FUNCTION_BLOCK WOOD_COUNTER
  {SET_ATTRIBUTE(OpcUa, SERVICE)}
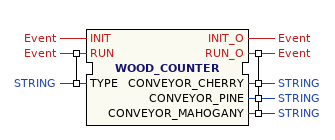
  EVENT_INPUT
    INIT;
    RUN WITH TYPE; {SET_ATTRIBUTE(OpcUa, Method)}
  END_EVENT
  EVENT_OUTPUT
    INIT_O;
    RUN_O WITH CONVEYOR_CHERRY, CONVEYOR_PINE, CONVEYOR_MAHOGANY;
  END_EVENT
  VAR_INPUT
    TYPE : STRING;
  END_VAR
  VAR_OUTPUT
    CONVEYOR_CHERRY : STRING;
    CONVEYOR_PINE : STRING;
    CONVEYOR_MAHOGANY : STRING;
  END_VAR
END_FUNCTION_BLOCK
